ADAPTER IDedicatedBlower (* Adapter Interface *)
  (* Standard: 61499-1 *)
  (* Version 0.0, 11/15/2023, SESA371406, Schneider Electric *)
  PACKAGE SE.Nereda;
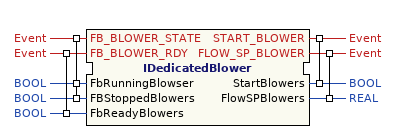
  EVENT_INPUT
    FB_BLOWER_STATE WITH FbRunningBlowser, FBStoppedBlowers;
    FB_BLOWER_RDY WITH FbReadyBlowers;
  END_EVENT
  EVENT_OUTPUT
    START_BLOWER WITH StartBlowers;
    FLOW_SP_BLOWER WITH FlowSPBlowers;
  END_EVENT
  VAR_INPUT
    FbRunningBlowser : BOOL;
    FBStoppedBlowers : BOOL;
    FbReadyBlowers : BOOL;
  END_VAR
  VAR_OUTPUT
    StartBlowers : BOOL;
    FlowSPBlowers : REAL;
  END_VAR
  SERVICE SOCKET/PLUG
    SEQUENCE request_confirm
      SOCKET.REQ(REQD) -> PLUG.REQ(REQD);
      PLUG.CNF(CNFD) -> SOCKET.CNF(CNFD);
    END_SEQUENCE
    SEQUENCE indication_response
      PLUG.IND(INDD) -> SOCKET.IND(INDD);
      SOCKET.RSP(RSPD) -> PLUG.RSP(RSPD);
    END_SEQUENCE
  END_SERVICE
END_ADAPTER
